FUNCTION_BLOCK FB_SQUARE
VAR_INPUT
	T_ON	:LREAL;//s
	T_OFF	:LREAL;//s
END_VAR
VAR_OUTPUT
	SQUARE:BOOL;
END_VAR
VAR
	Ton1,Ton2:TON;
	step:INT;
END_VAR

ton1(IN:=NOT SQUARE, PT:= LREAL_TO_TIME(T_OFF*1000), Q=> , ET=> );
ton2(IN:=  SQUARE, PT:=LREAL_TO_TIME(T_ON*1000) , Q=> , ET=> );
IF ton1.Q OR ton2.Q THEN
	SQUARE:=NOT SQUARE;
END_IF

END_FUNCTION_BLOCK

(* stored: Version 1.1.0.1, ProductVersion 3.1.4024.11
   POU FB_SQUARE: Id {8649238c-b769-431e-8960-5afaa1b59395}, SpecialFunc None *)
